// TIA Portal V19 export
TYPE "C402_VAR_IF_AFS_TYPIC"
   STRUCT
      STS_VKL_OK { ExternalAccessible := 'False'; ExternalVisible := 'False'; ExternalWritable := 'False'} : Bool;   // TRUE = verkeerslichten op rood, vrijgave sluiten afsluitbomen
      STS_VKL_AAN { ExternalAccessible := 'False'; ExternalVisible := 'False'; ExternalWritable := 'False'} : Bool;   // TRUE = verkeerslichten aangestuurd
      STS_KST_OPEN { ExternalAccessible := 'False'; ExternalVisible := 'False'; ExternalWritable := 'False'} : Bool;   // TRUE = deur wegkantkast geopend
      STO { ExternalAccessible := 'False'; ExternalVisible := 'False'; ExternalWritable := 'False'} : Struct   // Opsomming van alle signaleringen
         A001 : Bool;   // Noodstop
         A002 : Bool;   // Storing UPS
         A003 : Bool;   // UPS in batterijwerking
         A004 : Bool;   // Storing klimaatregeling wegkantkast
      END_STRUCT;
   END_STRUCT;
END_TYPE
